TYPE Piano450LaserConfig EXTENDS DeviceConfiguration :
STRUCT
	SerialCommunication : SerialCommunication;
END_STRUCT
END_TYPE

(* stored: Version 1.1.0.1, ProductVersion 3.1.4024.12
   DUT Piano450LaserConfig: Id {bb0995f0-1d95-42bf-a0ef-6e287716b99f} *)
